Fanuc KAREL source: CA0001.KL

-- PROVISIONAL review KL for V1013-1; original PC SHA256 92382ac1517bb574fd50c6e3344e38c4de6e4150d5008530e06574e2f3ac05a8
-- Incomplete behavior may be omitted. Consult companion uncertainty JSON. Do not deploy.
PROGRAM CA0001
%NOLOCKGROUP
VAR
  G : INTEGER
  I : INTEGER
  R : REAL
  B : BOOLEAN
  S : STRING[16]
-- UNRESOLVED_DECL AI type=002010
-- UNRESOLVED_DECL AR type=002011
-- UNRESOLVED_DECL ST type=001100
-- UNRESOLVED_DECL P type=000102
-- UNRESOLVED_DECL V type=000013
BEGIN
  -- UNRESOLVED_PC offsets 0-1; opcodes 7B
  -- UNRESOLVED_PC offsets 6-20; opcodes 21,9D,52,23
  -- UNRESOLVED_PC offsets 25-29; opcodes 7F
  -- UNRESOLVED_PC offsets 34-41; opcodes 9C,23
  -- UNRESOLVED_PC offsets 46-53; opcodes 9D,23
  -- UNRESOLVED_PC offsets 58-69; opcodes 2E,23
  -- UNRESOLVED_PC offsets 74-81; opcodes 9D,23
  -- UNRESOLVED_PC offsets 86-95; opcodes 3F,75
  -- UNRESOLVED_PC offsets 100-114; opcodes 2E,22,9D,33,35
  -- UNRESOLVED_PC offsets 119-133; opcodes 2E,22,9D,33,35
  -- UNRESOLVED_PC offsets 138-153; opcodes 2E,22,32,35
  -- UNRESOLVED_PC offsets 158-173; opcodes 2E,22,32,35
  -- UNRESOLVED_PC offsets 178-182; opcodes 27,AA
  -- UNRESOLVED_PC offsets 187-191; opcodes 7F
END CA0001
